FUNCTION_BLOCK FB_TCP_IP_ServerAccept
VAR_INPUT
	sSrvNetId: T_AmsNetId;
	bAccept: BOOL;
	bListenReady: BOOL;
	hListener: Tc2_TcpIp.T_HSOCKET;
	bSend: BOOL;
	bClose: BOOL;
	bReset: BOOL;
	aSendDataBuffer: ARRAY[0..MAX_BUFFER] OF BYTE;	
	TIMEOUT: TIME := T#5S;
	
END_VAR
VAR_OUTPUT
	//bDone: BOOL;
	//bBusy: BOOL;
	bAccepted: BOOL;
	bError: BOOL;
	nErrID: UDINT;
	sStatus: STRING(255);
	aReceiveDataBuffer: ARRAY[0..MAX_BUFFER] OF BYTE;
END_VAR
VAR
	step: (eInit, ePreAccept, eAccept, eManageConnection, eWait, ePreSend, eSend, eClose, eClose2, eCloseAll, eError);
	fbSocketAccept: FB_SocketAccept;
	fbSocketClose: FB_SocketClose;
	fbSocketSend: FB_SocketSend;
	fbSocketReceive: FB_SocketReceive;
	aDataBuffer: ARRAY[0..MAX_BUFFER] OF BYTE;
	nRecBytes: UDINT;

	rtSend: R_TRIG;
	rtClose: R_TRIG;
	tonReceivePollFreq: TON;
	rtReset: R_TRIG;
	tonError: TON;
	
	M_Close: BOOL;
	tonCloseCmdOverride: TON;
	M_Reset: BOOL;
	tonResetCmdOverride: TON;
	//tonCaseStuck: TON;
	tonAutoErrorReset: TON;
	nBytesTransferred: UDINT;
END_VAR
VAR CONSTANT
	MAX_BUFFER	: UINT:= 1023;
END_VAR

	rtClose(CLK:= bClose, Q=> );
	IF rtClose.Q THEN
		M_Close			:=	TRUE;
	END_IF
	tonCloseCmdOverride(IN:= M_Close, PT:= TIMEOUT + T#1S, Q=> , ET=> );
	IF tonCloseCmdOverride.Q THEN
		step		:=	eClose;
		M_Close		:=	FALSE;			
	END_IF

	rtReset(CLK:= bReset, Q=> );
	IF rtReset.Q THEN
		M_Reset			:=	TRUE;
	END_IF
	
//	IF bDone AND tonResetCmdOverride.Q THEN
//		step		:=	eInit;
//		M_Reset		:=	FALSE;
//		bDone		:=	FALSE;	
//	END_IF
	tonResetCmdOverride(IN:= M_Reset, PT:= TIMEOUT + T#1S, Q=> , ET=> );
	IF tonResetCmdOverride.Q THEN
		//bDone		:=	TRUE;	
		step		:=	eInit;
		M_Reset		:=	FALSE;	
	END_IF

	CASE step OF
	eInit:
		IF bAccept AND (bListenReady AND hListener.handle <> 0) AND (NOT bReset) AND (NOT bClose) THEN
			step		:=	ePreAccept;
			bAccepted	:=	FALSE;
		ELSIF M_Close AND (NOT bReset) THEN
			step		:=	eClose;
			M_Close		:=	FALSE;
		END_IF
		fbSocketAccept(bExecute:= FALSE);
		fbSocketClose(bExecute:= FALSE);
		fbSocketSend(bExecute:= FALSE);
		M_Reset			:=	FALSE;
		
	ePreAccept:
		fbSocketAccept(
			sSrvNetId		:= sSrvNetId, 
			hListener		:= hListener, 
			bExecute		:= TRUE, 
			tTimeout		:= TIMEOUT, 
			bAccepted		=> , 
			bBusy			=> , 
			bError			=> , 
			nErrId			=> , 
			hSocket			=> );
	
		IF fbSocketAccept.bError THEN
			step		:=	eError;
			nErrID		:=	fbSocketAccept.nErrId;
			sStatus		:=	'FB Error: fbSocketAccept | case no. ePreAccept';
		ELSE			
		//ELSIF (fbSocketAccept.bBusy) THEN	- Note: Observed that this FB does not trigger Busy bit
			step		:=	eAccept;
		END_IF

	eAccept:
		fbSocketAccept(
			sSrvNetId		:= sSrvNetId, 
			hListener		:= hListener, 
			bExecute		:= TRUE, 
			tTimeout		:= TIMEOUT, 
			bAccepted		=> , 
			bBusy			=> , 
			bError			=> , 
			nErrId			=> , 
			hSocket			=> );
			
		IF fbSocketAccept.bError THEN
			step		:=	eError;
			nErrID		:=	fbSocketAccept.nErrId;
			sStatus		:=	'FB Error: fbSocketAccept | case no. eAccept';
		ELSIF (NOT fbSocketAccept.bBusy) THEN
			IF fbSocketAccept.hSocket.handle <> 0 THEN
				step			:=	eManageConnection;
				bAccepted		:=	fbSocketAccept.bAccepted;
			ELSE
				step			:=	eManageConnection;
			END_IF	
			bError		:=	FALSE;
			nErrID		:=	0;
			sStatus		:=	'';
		END_IF	

	eManageConnection:
		IF NOT bAccepted THEN
			step		:=	eInit;
		ELSE
			step		:=	eWait;
		END_IF
	
	eWait:	
		IF rtSend.Q THEN
			step		:=	ePreSend;
		END_IF
		IF M_Close THEN
			M_Close		:=	FALSE;
			step		:=	eClose;
		END_IF
	
	ePreSend:
		fbSocketSend(
			sSrvNetId		:= sSrvNetId, 
			hSocket			:= fbSocketAccept.hSocket, 
			cbLen			:= SIZEOF(aSendDataBuffer), 
			pSrc			:= ADR(aSendDataBuffer), 
			bExecute		:= TRUE, 
			tTimeout		:= TIMEOUT, 
			bBusy			=> , 
			bError			=> , 
			nErrId			=> );	
	
		IF fbSocketSend.bError THEN
			step			:=	eError;
			nErrID			:=	fbSocketSend.nErrId;
			sStatus			:=	'FB_SocketSend | error case: ePreSend';
		ELSIF (fbSocketSend.bBusy) THEN
			fbSocketSend(bExecute	:=	FALSE);
			step			:=	eSend;		
		END_IF			
		
	eSend:
		fbSocketSend(
			sSrvNetId		:= sSrvNetId, 
			hSocket			:= fbSocketAccept.hSocket, 
			cbLen			:= SIZEOF(aSendDataBuffer), 
			pSrc			:= ADR(aSendDataBuffer), 
			bExecute		:= TRUE, 
			tTimeout		:= TIMEOUT, 
			bBusy			=> , 
			bError			=> , 
			nErrId			=> );	
	
		IF fbSocketSend.bError THEN
			step			:=	eError;
			nErrID			:=	fbSocketSend.nErrId;
			sStatus			:=	'FB_SocketSend | error case: eSend';
		ELSIF (NOT fbSocketSend.bBusy) THEN
			fbSocketSend(bExecute	:=	FALSE);
			step			:=	eWait;		
		END_IF	
		
	eClose:		
		bAccepted			:=	FALSE;
		
		fbSocketClose(
			sSrvNetId		:= sSrvNetId, 
			hSocket			:= fbSocketAccept.hSocket, 
			bExecute		:= TRUE, 
			tTimeout		:= TIMEOUT, 
			bBusy			=> , 
			bError			=> , 
			nErrId			=> );
			
		IF fbSocketClose.bError THEN
			step		:=	eError;
			nErrID		:=	fbSocketClose.nErrId;
			sStatus		:=	'FB Error: fbSocketClose | case no. eClose';			
		ELSIF (NOT fbSocketClose.bBusy) THEN
			step		:=	eClose2;
		END_IF	
	
	eClose2:

		fbSocketClose(
			sSrvNetId		:= sSrvNetId, 
			hSocket			:= fbSocketAccept.hListener, 
			bExecute		:= TRUE, 
			tTimeout		:= TIMEOUT, 
			bBusy			=> , 
			bError			=> , 
			nErrId			=> );
			
		IF fbSocketClose.bError THEN
			step		:=	eError;
			nErrID		:=	fbSocketClose.nErrId;
			sStatus		:=	'FB Error: fbSocketClose | case no. eClose';			
		ELSIF (NOT fbSocketClose.bBusy) THEN
			fbSocketClose(bExecute:= FALSE);
			step		:=	eInit;

		END_IF	
		
	eError:
		bError		:=	TRUE;
		//bBusy		:=	FALSE;
		//bDone		:=	FALSE;
		
		bAccepted	:=	FALSE;
		fbSocketAccept(bExecute:= FALSE);
		fbSocketClose(bExecute:= FALSE);
		fbSocketSend(bExecute:= FALSE);
		
		tonAutoErrorReset(IN:= bAccept, PT:= T#5S, Q=> , ET=> );
		IF tonAutoErrorReset.Q THEN
			step	:=	eInit;
			tonAutoErrorReset(IN:= FALSE);			
		END_IF
		
		IF M_Close THEN
			step	:=	eClose;
			M_Close	:=	FALSE;
			tonAutoErrorReset(IN:= FALSE);
			bError		:=	FALSE;
			nErrID		:=	0;
			sStatus		:=	'';
		ELSIF M_Reset THEN
			step	:=	eInit;
			M_Reset	:=	FALSE;
			tonAutoErrorReset(IN:= FALSE);
			bError		:=	FALSE;
			nErrID		:=	0;
			sStatus		:=	'';	
		END_IF
		
	END_CASE
	
	tonReceivePollFreq(IN:= (NOT tonReceivePollFreq.Q) AND 
							bAccepted AND 
							(NOT bError) AND 
							(NOT fbSocketReceive.bBusy), 
						PT:= T#1S, Q=> , ET=> );
	
		fbSocketReceive(
			sSrvNetId		:= sSrvNetId, 
			hSocket			:= fbSocketAccept.hSocket, 
			cbLen			:= SIZEOF(aDataBuffer), 
			pDest			:= ADR(aDataBuffer), 
			bExecute		:= tonReceivePollFreq.Q, 
			tTimeout		:= TIMEOUT, 
			bBusy			=> , 
			bError			=> , 
			nErrId			=> , 
			nRecBytes		=> nRecBytes);	
		
		IF fbSocketReceive.nRecBytes > 0 THEN			
			FN_MemoryClear(destAddr:= ADR(aReceiveDataBuffer), Len:= SIZEOF(aReceiveDataBuffer));
		
			nBytesTransferred	:=	MEMCPY(destAddr:= ADR(aReceiveDataBuffer), srcAddr:= ADR(aDataBuffer), n:= nRecBytes);
			IF (nRecBytes <> nBytesTransferred) AND step = eWait THEN
				bError		:=	TRUE;
				nErrID		:=	1;
				sStatus		:=	'Bytes transfered is nt equal to received bytes | Custom Error ID';
				step		:=	eError;
			END_IF
		END_IF

END_FUNCTION_BLOCK

(* stored: Version 1.1.0.1, ProductVersion 3.1.4024.13
   POU FB_TCP_IP_ServerAccept: Id {4b0e0506-87dd-4ff1-980f-9e1f09a2edf7}, SpecialFunc None *)
